{attribute 'qualified_only'}
VAR_GLOBAL
	tTaskCycleTime			: TIME := T#50MS;
END_VAR

(* stored: Version 1.1.0.1, ProductVersion 3.1.4024.10
   GVL GlobalVariables: Id {03b0febb-bd51-42dd-a1dc-b1b77f4022cb} *)
